FUNCTION_BLOCK FB_TestFunctionBlock
VAR
	nCounter : LINT;
END_VAR

nCounter := nCounter + 1;

END_FUNCTION_BLOCK

(* stored: Version 1.1.0.1, ProductVersion 3.1.4024.12
   POU FB_TestFunctionBlock: Id {b0a54a4d-cef1-4465-aa75-b643b5e47f92}, SpecialFunc None *)
